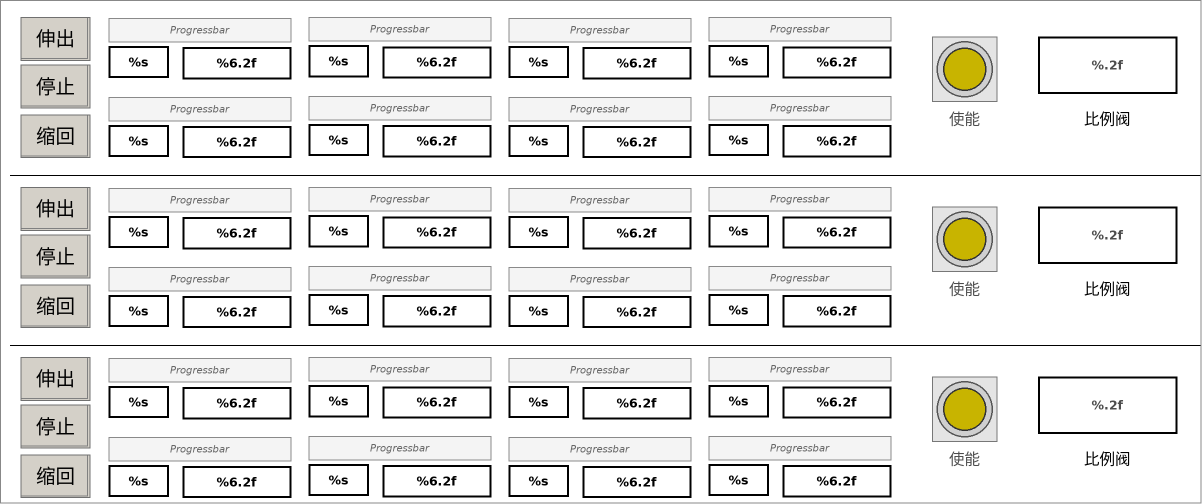
VISUALIZATION Ceiling_Rail_345  // 1202x504
    Frame (3,6 892x156)
        shows ModuleX8(extendButton := gUI.TiG.arrPV[3].sColumn[1].bExtend, retractButton := gUI.TiG.arrPV[3].sColumn[1].bRetract, stopButton := gUI.TiG.arrPV[3].sColumn[1].bStop, nameStr1 := gUI.TiG.arrPV[3].sNum[1].strName, posVal1 := gUI.TiG.arrPV[3].sNum[1].rPosition, percentBar1 := gUI.TiG.arrPV[3].sNum[1].rPercent, nameStr2 := gUI.TiG.arrPV[3].sNum[2].strName, posVal2 := gUI.TiG.arrPV[3].sNum[2].rPosition, percentBar2 := gUI.TiG.arrPV[3].sNum[2].rPercent, nameStr3 := gUI.TiG.arrPV[3].sNum[3].strName, posVal3 := gUI.TiG.arrPV[3].sNum[3].rPosition, percentBar3 := gUI.TiG.arrPV[3].sNum[3].rPercent, nameStr4 := gUI.TiG.arrPV[3].sNum[4].strName, posVal4 := gUI.TiG.arrPV[3].sNum[4].rPosition, percentBar4 := gUI.TiG.arrPV[3].sNum[4].rPercent, nameStr5 := gUI.TiG.arrPV[3].sNum[5].strName, posVal5 := gUI.TiG.arrPV[3].sNum[5].rPosition, percentBar5 := gUI.TiG.arrPV[3].sNum[5].rPercent, nameStr6 := gUI.TiG.arrPV[3].sNum[6].strName, posVal6 := gUI.TiG.arrPV[3].sNum[6].rPosition, percentBar6 := gUI.TiG.arrPV[3].sNum[6].rPercent, nameStr7 := gUI.TiG.arrPV[3].sNum[7].strName, posVal7 := gUI.TiG.arrPV[3].sNum[7].rPosition, percentBar7 := gUI.TiG.arrPV[3].sNum[7].rPercent, nameStr8 := gUI.TiG.arrPV[3].sNum[8].strName, posVal8 := gUI.TiG.arrPV[3].sNum[8].rPosition, percentBar8 := gUI.TiG.arrPV[3].sNum[8].rPercent)
    Frame (3,176 892x156)
        shows ModuleX8(extendButton := gUI.TiG.arrPV[4].sColumn[1].bExtend, retractButton := gUI.TiG.arrPV[4].sColumn[1].bRetract, stopButton := gUI.TiG.arrPV[4].sColumn[1].bStop, nameStr1 := gUI.TiG.arrPV[4].sNum[1].strName, posVal1 := gUI.TiG.arrPV[4].sNum[1].rPosition, percentBar1 := gUI.TiG.arrPV[4].sNum[1].rPercent, nameStr2 := gUI.TiG.arrPV[4].sNum[2].strName, posVal2 := gUI.TiG.arrPV[4].sNum[2].rPosition, percentBar2 := gUI.TiG.arrPV[4].sNum[2].rPercent, nameStr3 := gUI.TiG.arrPV[4].sNum[3].strName, posVal3 := gUI.TiG.arrPV[4].sNum[3].rPosition, percentBar3 := gUI.TiG.arrPV[4].sNum[3].rPercent, nameStr4 := gUI.TiG.arrPV[4].sNum[4].strName, posVal4 := gUI.TiG.arrPV[4].sNum[4].rPosition, percentBar4 := gUI.TiG.arrPV[4].sNum[4].rPercent, nameStr5 := gUI.TiG.arrPV[4].sNum[5].strName, posVal5 := gUI.TiG.arrPV[4].sNum[5].rPosition, percentBar5 := gUI.TiG.arrPV[4].sNum[5].rPercent, nameStr6 := gUI.TiG.arrPV[4].sNum[6].strName, posVal6 := gUI.TiG.arrPV[4].sNum[6].rPosition, percentBar6 := gUI.TiG.arrPV[4].sNum[6].rPercent, nameStr7 := gUI.TiG.arrPV[4].sNum[7].strName, posVal7 := gUI.TiG.arrPV[4].sNum[7].rPosition, percentBar7 := gUI.TiG.arrPV[4].sNum[7].rPercent, nameStr8 := gUI.TiG.arrPV[4].sNum[8].strName, posVal8 := gUI.TiG.arrPV[4].sNum[8].rPosition, percentBar8 := gUI.TiG.arrPV[4].sNum[8].rPercent)
    Frame (3,346 892x156)
        shows ModuleX8(extendButton := gUI.TiG.arrPV[5].sColumn[1].bExtend, retractButton := gUI.TiG.arrPV[5].sColumn[1].bRetract, stopButton := gUI.TiG.arrPV[5].sColumn[1].bStop, nameStr1 := gUI.TiG.arrPV[5].sNum[1].strName, posVal1 := gUI.TiG.arrPV[5].sNum[1].rPosition, percentBar1 := gUI.TiG.arrPV[5].sNum[1].rPercent, nameStr2 := gUI.TiG.arrPV[5].sNum[2].strName, posVal2 := gUI.TiG.arrPV[5].sNum[2].rPosition, percentBar2 := gUI.TiG.arrPV[5].sNum[2].rPercent, nameStr3 := gUI.TiG.arrPV[5].sNum[3].strName, posVal3 := gUI.TiG.arrPV[5].sNum[3].rPosition, percentBar3 := gUI.TiG.arrPV[5].sNum[3].rPercent, nameStr4 := gUI.TiG.arrPV[5].sNum[4].strName, posVal4 := gUI.TiG.arrPV[5].sNum[4].rPosition, percentBar4 := gUI.TiG.arrPV[5].sNum[4].rPercent, nameStr5 := gUI.TiG.arrPV[5].sNum[5].strName, posVal5 := gUI.TiG.arrPV[5].sNum[5].rPosition, percentBar5 := gUI.TiG.arrPV[5].sNum[5].rPercent, nameStr6 := gUI.TiG.arrPV[5].sNum[6].strName, posVal6 := gUI.TiG.arrPV[5].sNum[6].rPosition, percentBar6 := gUI.TiG.arrPV[5].sNum[6].rPercent, nameStr7 := gUI.TiG.arrPV[5].sNum[7].strName, posVal7 := gUI.TiG.arrPV[5].sNum[7].rPosition, percentBar7 := gUI.TiG.arrPV[5].sNum[7].rPercent, nameStr8 := gUI.TiG.arrPV[5].sNum[8].strName, posVal8 := gUI.TiG.arrPV[5].sNum[8].rPosition, percentBar8 := gUI.TiG.arrPV[5].sNum[8].rPercent)
    Frame (918,31 261x106)
        shows ModuleDTD(enable := gUI.TiG.arrPV[3].bPVD_enable, propPercent := gUI.TiG.arrPV[3].rPVDPercent)
    Frame (918,201 261x106)
        shows ModuleDTD(enable := gUI.TiG.arrPV[4].bPVD_enable, propPercent := gUI.TiG.arrPV[4].rPVDPercent)
    Frame (918,371 261x106)
        shows ModuleDTD(enable := gUI.TiG.arrPV[5].bPVD_enable, propPercent := gUI.TiG.arrPV[5].rPVDPercent)
    Line (10,175) (1200,175)
    Line (10,345) (1200,345)
END_VISUALIZATION

// Device/Application/display/OrigTi/Ceiling_Rail6
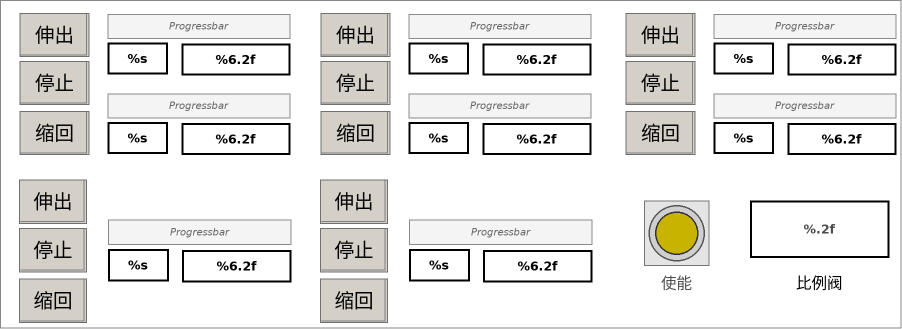
VISUALIZATION Ceiling_Rail6  // 902x329
    Frame (2,169 293x158)
        shows ModuleX1(extendButton := gUI.TiG.arrPV[6].sColumn[2].bExtend, retractButton := gUI.TiG.arrPV[6].sColumn[2].bRetract, stopButton := gUI.TiG.arrPV[6].sColumn[2].bStop, nameStr := gUI.TiG.arrPV[6].sNum[3].strName, posVal := gUI.TiG.arrPV[6].sNum[3].rPosition, percentBar := gUI.TiG.arrPV[6].sNum[3].rPercent)
    Frame (2,3 292x156)
        shows ModuleX2(extendButton := gUI.TiG.arrPV[6].sColumn[1].bExtend, retractButton := gUI.TiG.arrPV[6].sColumn[1].bRetract, stopButton := gUI.TiG.arrPV[6].sColumn[1].bStop, nameStr1 := gUI.TiG.arrPV[6].sNum[1].strName, posVal1 := gUI.TiG.arrPV[6].sNum[1].rPosition, percentBar1 := gUI.TiG.arrPV[6].sNum[1].rPercent, nameStr2 := gUI.TiG.arrPV[6].sNum[2].strName, posVal2 := gUI.TiG.arrPV[6].sNum[2].rPosition, percentBar2 := gUI.TiG.arrPV[6].sNum[2].rPercent)
    Frame (303,3 292x156)
        shows ModuleX2(extendButton := gUI.TiG.arrPV[6].sColumn[3].bExtend, retractButton := gUI.TiG.arrPV[6].sColumn[3].bRetract, stopButton := gUI.TiG.arrPV[6].sColumn[3].bStop, nameStr1 := gUI.TiG.arrPV[6].sNum[4].strName, posVal1 := gUI.TiG.arrPV[6].sNum[4].rPosition, percentBar1 := gUI.TiG.arrPV[6].sNum[4].rPercent, nameStr2 := gUI.TiG.arrPV[6].sNum[5].strName, posVal2 := gUI.TiG.arrPV[6].sNum[5].rPosition, percentBar2 := gUI.TiG.arrPV[6].sNum[5].rPercent)
    Frame (303,169 293x158)
        shows ModuleX1(extendButton := gUI.TiG.arrPV[6].sColumn[4].bExtend, retractButton := gUI.TiG.arrPV[6].sColumn[4].bRetract, stopButton := gUI.TiG.arrPV[6].sColumn[4].bStop, nameStr := gUI.TiG.arrPV[6].sNum[6].strName, posVal := gUI.TiG.arrPV[6].sNum[6].rPosition, percentBar := gUI.TiG.arrPV[6].sNum[6].rPercent)
    Frame (608,3 292x156)
        shows ModuleX2(extendButton := gUI.TiG.arrPV[6].sColumn[5].bExtend, retractButton := gUI.TiG.arrPV[6].sColumn[5].bRetract, stopButton := gUI.TiG.arrPV[6].sColumn[5].bStop, nameStr1 := gUI.TiG.arrPV[6].sNum[7].strName, posVal1 := gUI.TiG.arrPV[6].sNum[7].rPosition, percentBar1 := gUI.TiG.arrPV[6].sNum[7].rPercent, nameStr2 := gUI.TiG.arrPV[6].sNum[8].strName, posVal2 := gUI.TiG.arrPV[6].sNum[8].rPosition, percentBar2 := gUI.TiG.arrPV[6].sNum[8].rPercent)
    Frame (630,195 261x106)
        shows ModuleDTD(enable := gUI.TiG.arrPV[6].bPVD_enable, propPercent := gUI.TiG.arrPV[6].rPVDPercent)
END_VISUALIZATION

// Device/Application/display/OrigTi/Ceiling_Rail7
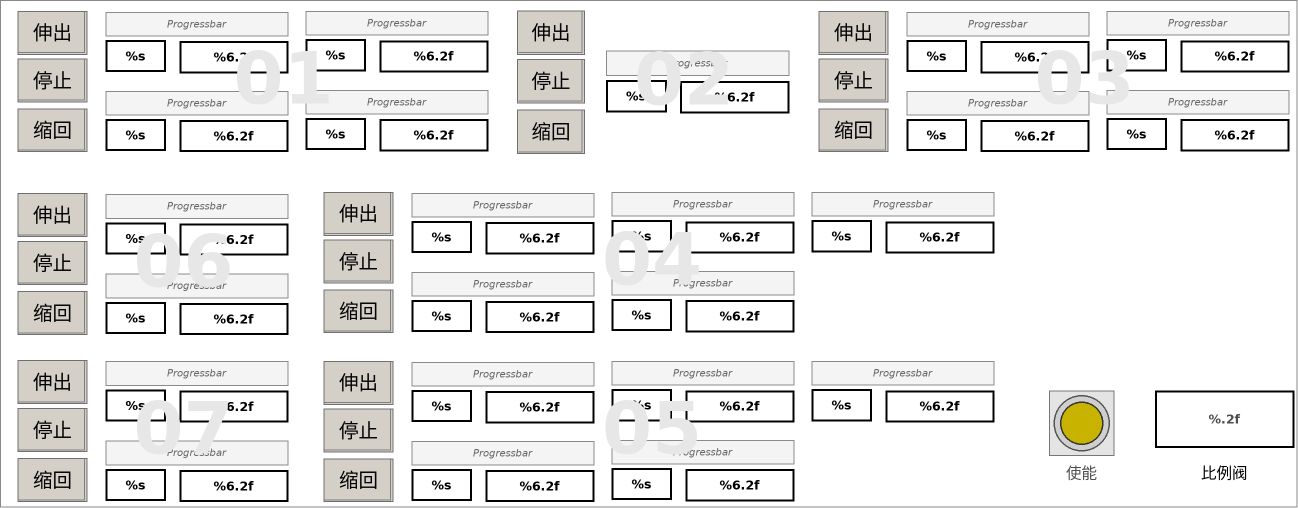
VISUALIZATION Ceiling_Rail7  // 1298x508
    Frame (0,0 492x156), "01"
        shows ModuleX4(extendButton := gUI.TiG.arrPV[7].sColumn[1].bExtend, retractButton := gUI.TiG.arrPV[7].sColumn[1].bRetract, stopButton := gUI.TiG.arrPV[7].sColumn[1].bStop, nameStr1 := gUI.TiG.arrPV[7].sNum[1].strName, posVal1 := gUI.TiG.arrPV[7].sNum[1].rPosition, percentBar1 := gUI.TiG.arrPV[7].sNum[1].rPercent, nameStr2 := gUI.TiG.arrPV[7].sNum[2].strName, posVal2 := gUI.TiG.arrPV[7].sNum[2].rPosition, percentBar2 := gUI.TiG.arrPV[7].sNum[2].rPercent, nameStr3 := gUI.TiG.arrPV[7].sNum[3].strName, posVal3 := gUI.TiG.arrPV[7].sNum[3].rPosition, percentBar3 := gUI.TiG.arrPV[7].sNum[3].rPercent, nameStr4 := gUI.TiG.arrPV[7].sNum[4].strName, posVal4 := gUI.TiG.arrPV[7].sNum[4].rPosition, percentBar4 := gUI.TiG.arrPV[7].sNum[4].rPercent)
    Frame (500,0 293x158), "02"
        shows ModuleX1(extendButton := gUI.TiG.arrPV[7].sColumn[2].bExtend, retractButton := gUI.TiG.arrPV[7].sColumn[2].bRetract, stopButton := gUI.TiG.arrPV[7].sColumn[2].bStop, nameStr := gUI.TiG.arrPV[7].sNum[5].strName, posVal := gUI.TiG.arrPV[7].sNum[5].rPosition, percentBar := gUI.TiG.arrPV[7].sNum[5].rPercent)
    Frame (801,0 492x156), "03"
        shows ModuleX4(extendButton := gUI.TiG.arrPV[7].sColumn[3].bExtend, retractButton := gUI.TiG.arrPV[7].sColumn[3].bRetract, stopButton := gUI.TiG.arrPV[7].sColumn[3].bStop, nameStr1 := gUI.TiG.arrPV[7].sNum[6].strName, posVal1 := gUI.TiG.arrPV[7].sNum[6].rPosition, percentBar1 := gUI.TiG.arrPV[7].sNum[6].rPercent, nameStr2 := gUI.TiG.arrPV[7].sNum[7].strName, posVal2 := gUI.TiG.arrPV[7].sNum[7].rPosition, percentBar2 := gUI.TiG.arrPV[7].sNum[7].rPercent, nameStr3 := gUI.TiG.arrPV[7].sNum[8].strName, posVal3 := gUI.TiG.arrPV[7].sNum[8].rPosition, percentBar3 := gUI.TiG.arrPV[7].sNum[8].rPercent, nameStr4 := gUI.TiG.arrPV[7].sNum[9].strName, posVal4 := gUI.TiG.arrPV[7].sNum[9].rPosition, percentBar4 := gUI.TiG.arrPV[7].sNum[9].rPercent)
    Frame (306,181 692x156), "04"
        shows ModuleX5(extendButton := gUI.TiG.arrPV[7].sColumn[4].bExtend, retractButton := gUI.TiG.arrPV[7].sColumn[4].bRetract, stopButton := gUI.TiG.arrPV[7].sColumn[4].bStop, nameStr1 := gUI.TiG.arrPV[7].sNum[10].strName, posVal1 := gUI.TiG.arrPV[7].sNum[10].rPosition, percentBar1 := gUI.TiG.arrPV[7].sNum[10].rPercent, nameStr2 := gUI.TiG.arrPV[7].sNum[11].strName, posVal2 := gUI.TiG.arrPV[7].sNum[11].rPosition, percentBar2 := gUI.TiG.arrPV[7].sNum[11].rPercent, nameStr3 := gUI.TiG.arrPV[7].sNum[12].strName, posVal3 := gUI.TiG.arrPV[7].sNum[12].rPosition, percentBar3 := gUI.TiG.arrPV[7].sNum[12].rPercent, nameStr4 := gUI.TiG.arrPV[7].sNum[13].strName, posVal4 := gUI.TiG.arrPV[7].sNum[13].rPosition, percentBar4 := gUI.TiG.arrPV[7].sNum[13].rPercent, nameStr5 := gUI.TiG.arrPV[7].sNum[14].strName, posVal5 := gUI.TiG.arrPV[7].sNum[14].rPosition, percentBar5 := gUI.TiG.arrPV[7].sNum[14].rPercent)
    Frame (306,350 692x156), "05"
        shows ModuleX5(extendButton := gUI.TiG.arrPV[7].sColumn[5].bExtend, retractButton := gUI.TiG.arrPV[7].sColumn[5].bRetract, stopButton := gUI.TiG.arrPV[7].sColumn[5].bStop, nameStr1 := gUI.TiG.arrPV[7].sNum[15].strName, posVal1 := gUI.TiG.arrPV[7].sNum[15].rPosition, percentBar1 := gUI.TiG.arrPV[7].sNum[15].rPercent, nameStr2 := gUI.TiG.arrPV[7].sNum[16].strName, posVal2 := gUI.TiG.arrPV[7].sNum[16].rPosition, percentBar2 := gUI.TiG.arrPV[7].sNum[16].rPercent, nameStr3 := gUI.TiG.arrPV[7].sNum[17].strName, posVal3 := gUI.TiG.arrPV[7].sNum[17].rPosition, percentBar3 := gUI.TiG.arrPV[7].sNum[17].rPercent, nameStr4 := gUI.TiG.arrPV[7].sNum[18].strName, posVal4 := gUI.TiG.arrPV[7].sNum[18].rPosition, percentBar4 := gUI.TiG.arrPV[7].sNum[18].rPercent, nameStr5 := gUI.TiG.arrPV[7].sNum[19].strName, posVal5 := gUI.TiG.arrPV[7].sNum[19].rPosition, percentBar5 := gUI.TiG.arrPV[7].sNum[19].rPercent)
    Frame (0,183 292x156), "06"
        shows ModuleX2(extendButton := gUI.TiG.arrPV[7].sColumn[6].bExtend, retractButton := gUI.TiG.arrPV[7].sColumn[6].bRetract, stopButton := gUI.TiG.arrPV[7].sColumn[6].bStop, nameStr1 := gUI.TiG.arrPV[7].sNum[20].strName, posVal1 := gUI.TiG.arrPV[7].sNum[20].rPosition, percentBar1 := gUI.TiG.arrPV[7].sNum[20].rPercent, nameStr2 := gUI.TiG.arrPV[7].sNum[21].strName, posVal2 := gUI.TiG.arrPV[7].sNum[21].rPosition, percentBar2 := gUI.TiG.arrPV[7].sNum[21].rPercent)
    Frame (0,350 292x156), "07"
        shows ModuleX2(extendButton := gUI.TiG.arrPV[7].sColumn[7].bExtend, retractButton := gUI.TiG.arrPV[7].sColumn[7].bRetract, stopButton := gUI.TiG.arrPV[7].sColumn[7].bStop, nameStr1 := gUI.TiG.arrPV[7].sNum[22].strName, posVal1 := gUI.TiG.arrPV[7].sNum[22].rPosition, percentBar1 := gUI.TiG.arrPV[7].sNum[22].rPercent, nameStr2 := gUI.TiG.arrPV[7].sNum[23].strName, posVal2 := gUI.TiG.arrPV[7].sNum[23].rPosition, percentBar2 := gUI.TiG.arrPV[7].sNum[23].rPercent)
    Frame (1035,385 261x106)
        shows ModuleDTD(enable := gUI.TiG.arrPV[7].bPVD_enable, propPercent := gUI.TiG.arrPV[7].rPVDPercent)
END_VISUALIZATION

// Device/Application/display/OrigTi/Ceiling_Rail_12
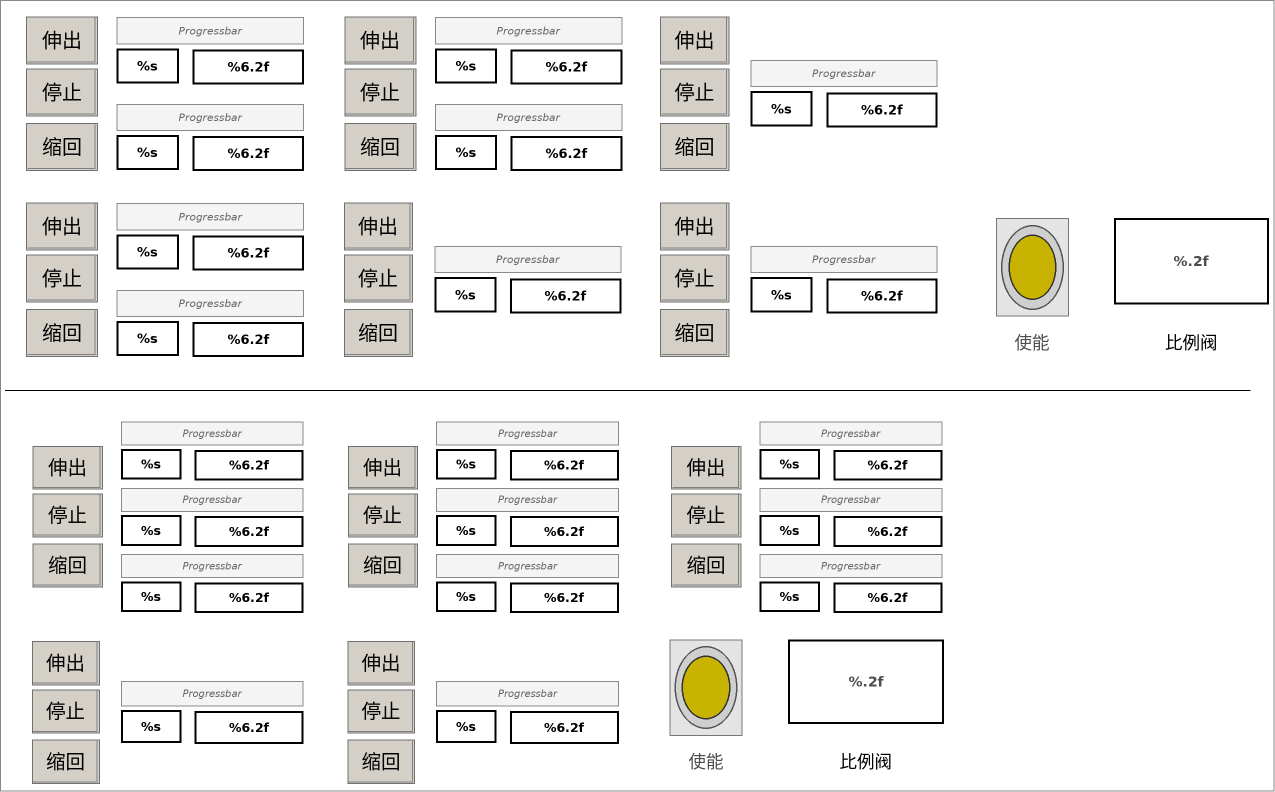
VISUALIZATION Ceiling_Rail_12  // 1275x792
    Line (5,390) (1250,390)
    Frame (3,0 1270x372)
        shows Ceiling_Rail1()
    Frame (2,403 946x387)
        shows Ceiling_Rail2()
END_VISUALIZATION

// Device/Application/display/OrigTi/Ceiling_Rail_67
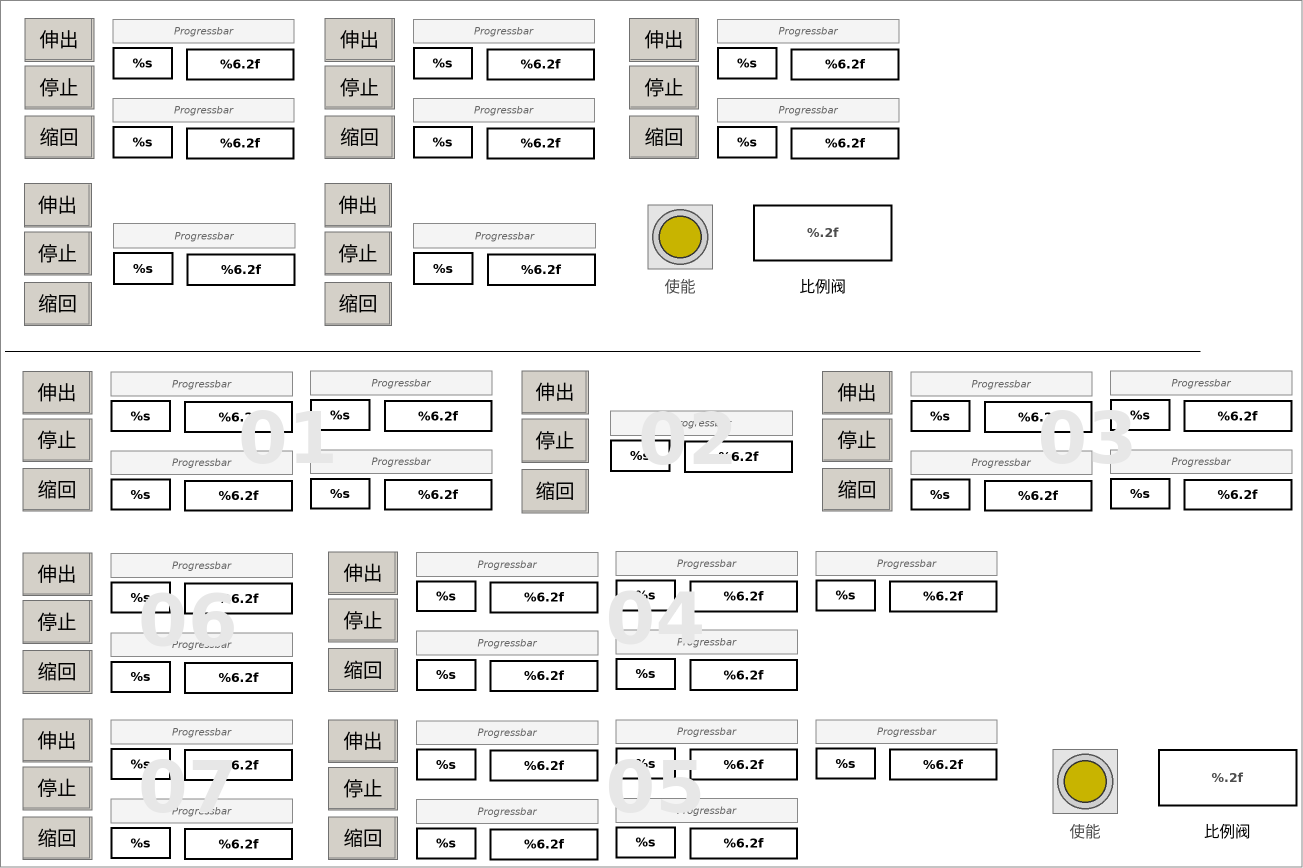
VISUALIZATION Ceiling_Rail_67  // 1303x868
    Line (5,351) (1200,351)
    Frame (5,5 900x327)
        shows Ceiling_Rail6()
    Frame (5,360 1296x506)
        shows Ceiling_Rail7()
END_VISUALIZATION

// Device/Application/display/Ceiling_Rail
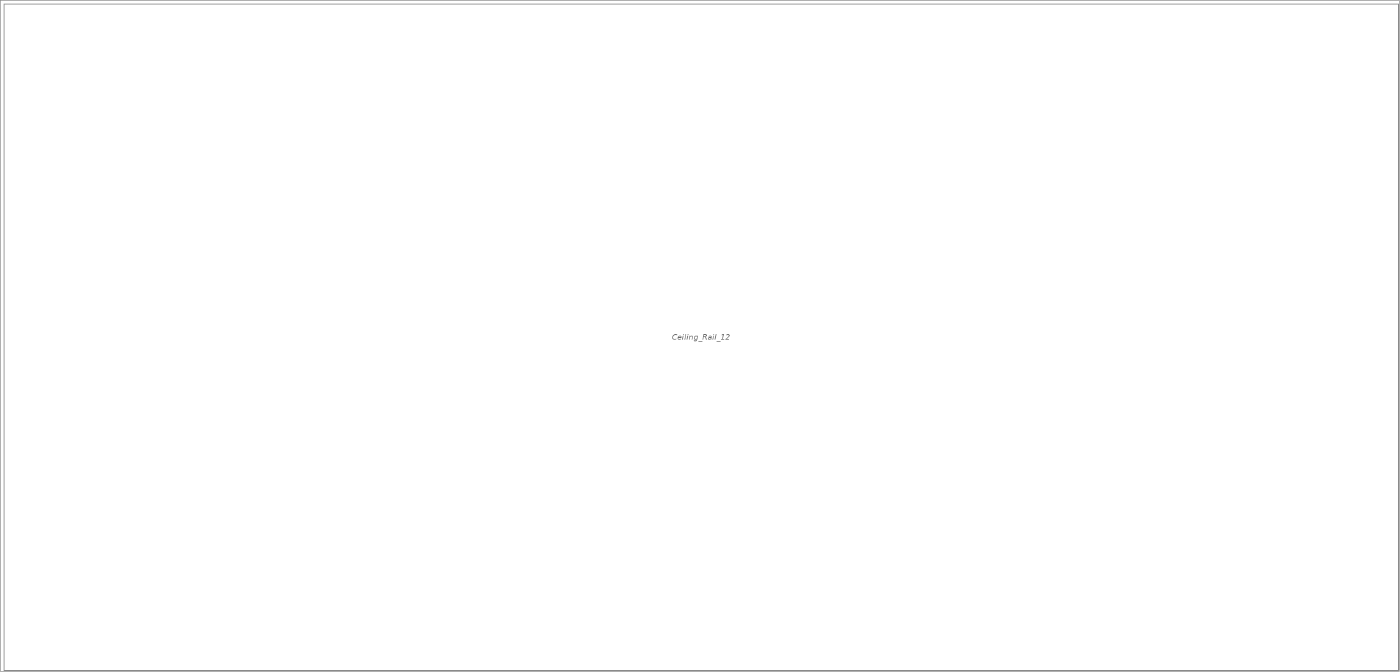
VISUALIZATION Ceiling_Rail  // 1847x887
    TabControl (5,5 1840x880)
        shows Ceiling_Rail_12()
        shows Ceiling_Rail_345()
        shows Ceiling_Rail_67()
        shows Ceiling_Rail_Plate()
        shows ManualMode()
        [0]: TabTitle=天轨1-2, ImageId=__VisualizationStyle.Element-Lamp-Lamp1-Blue-Off
        [1]: TabTitle=天轨3-5, ImageId=__VisualizationStyle.Element-Lamp-Lamp1-Blue-Off
        [2]: TabTitle=天轨6-7, ImageId=__VisualizationStyle.Element-Lamp-Lamp1-Blue-Off
        [3]: TabTitle=天轨挡板, ImageId=__VisualizationStyle.Element-Lamp-Lamp1-Blue-Off
        [4]: TabTitle=手动模式, ImageId=__VisualizationStyle.Element-Lamp-Lamp1-Blue-Off
END_VISUALIZATION

// Device/Application/display/OrigDi/Rotate_Plant
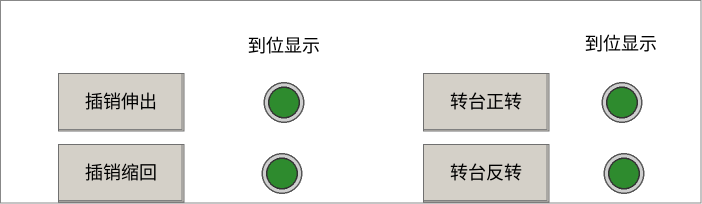
VISUALIZATION Rotate_Plant  // 702x204
    Button (58,73 126x58), "插销伸出"
        toggle gUI.TiG.sRot.oilExtend
    Button (58,144 126x58), "插销缩回"
        toggle gUI.TiG.sRot.oilRetract
    Button (423,73 126x58), "转台正转"
        toggle gUI.TiG.sRot.rotFront
    Button (423,144 126x58), "转台反转"
        toggle gUI.TiG.sRot.rotReverse
    Lamp1 (260,79 48x47), variable: gUI.TiG.sRotLed.oilExtended, style: Lamp-Lamp1-Green
    Lamp1 (258,150 48x47), variable: gUI.TiG.sRotLed.oilRetracted, style: Lamp-Lamp1-Green
    Lamp1 (598,79 48x47), variable: gUI.TiG.sRotLed.platExtended, style: Lamp-Lamp1-Green
    Lamp1 (600,150 48x47), variable: gUI.TiG.sRotLed.platRetracted, style: Lamp-Lamp1-Green
    Label (205,31 158x30), "到位显示"
    Label (542,29 158x30), "到位显示"
END_VISUALIZATION

// Device/Application/display/OrigTi/Ceiling_Rail_Plate
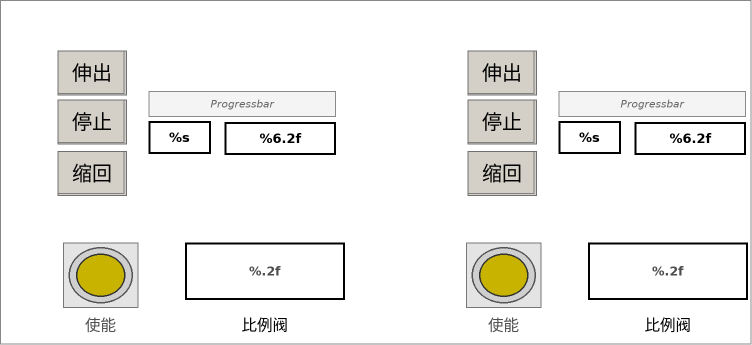
VISUALIZATION Ceiling_Rail_Plate  // 752x345
    Frame (40,40 300x160)
        shows ModuleX1(extendButton := gUI.TiG.arrPlate[1].sCmd.bExtend, retractButton := gUI.TiG.arrPlate[1].sCmd.bRetract, stopButton := gUI.TiG.arrPlate[1].sCmd.bStop, nameStr := gUI.TiG.arrPlate[1].sInfo.strName, posVal := gUI.TiG.arrPlate[1].sInfo.rPosition, percentBar := gUI.TiG.arrPlate[1].sInfo.rPercent)
    Frame (450,40 300x160)
        shows ModuleX1(extendButton := gUI.TiG.arrPlate[2].sCmd.bExtend, retractButton := gUI.TiG.arrPlate[2].sCmd.bRetract, stopButton := gUI.TiG.arrPlate[2].sCmd.bStop, nameStr := gUI.TiG.arrPlate[2].sInfo.strName, posVal := gUI.TiG.arrPlate[2].sInfo.rPosition, percentBar := gUI.TiG.arrPlate[2].sInfo.rPercent)
    Frame (47,237 300x106)
        shows ModuleDTD(enable := gUI.TiG.arrPV[6].bPVD_enable, propPercent := gUI.TiG.arrPV[6].rPVDPercent)
    Frame (450,237 300x106)
        shows ModuleDTD(enable := gUI.TiG.arrPV[1].bPVD_enable, propPercent := gUI.TiG.arrPV[1].rPVDPercent)
END_VISUALIZATION

// Device/Application/display/OrigTi/ManualMode
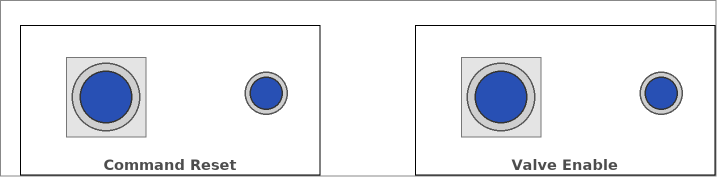
VISUALIZATION ManualMode  // 717x177
    Rectangle (20,25 300x150), "Command Reset"
    Lamp1 (241,68 50x50), variable: gUI.sManualMode.bCmdReset, style: Lamp-Lamp1-Blue
    PushSwitchLed (66,57 80x80), variable: gUI.sManualMode.bCmdReset, behaviour: TOGGLE, style: Switch-PushSwitchLed-Blue
    Rectangle (415,25 300x150), "Valve Enable"
    Lamp1 (636,68 50x50), variable: gUI.sManualMode.bDteEnable, style: Lamp-Lamp1-Blue
    PushSwitchLed (461,57 80x80), variable: gUI.sManualMode.bDteEnable, behaviour: TOGGLE, style: Switch-PushSwitchLed-Blue
END_VISUALIZATION
